	(*Robot At Home (Work Home or Intermediate Home)*)
	IF FB_In.Robot_Type=DX100
		THEN
		At_Home:= In_Cube64 OR In_Cube1 OR In_Cube2 OR In_Cube3 OR In_Cube4;
	ELSIF FB_In.Robot_Type=DX100_Dual
		THEN
		At_Home:= In_Cube64 OR In_Cube1 OR In_Cube2 OR In_Cube3 OR In_Cube4;
	ELSIF FB_In.Robot_Type=DX100_3_MIG
		THEN
		R1_At_Home:= R1_In_Cube64;
		R2_At_Home:= R2_In_Cube63;
		R3_At_Home:= R3_In_Cube62;
		At_Home:= R1_At_Home AND R2_At_Home AND R3_At_Home;
	ELSIF FB_In.Robot_Type=NX100
		THEN
		At_Home:= In_Cube32 OR In_Cube1 OR In_Cube2 OR In_Cube3 OR In_Cube4;
	ELSE
		At_Home:= In_Cube24 OR In_Cube1 OR In_Cube2 OR In_Cube3 OR In_Cube4;
	END_IF;
	(*At Equipment Interference Zones*)
	At_EquipInterf1:= NOT Clear_Of_EquipInterf1 AND Clear_Of_EquipInterf2 AND Clear_Of_EquipInterf3 AND Clear_Of_EquipInterf4
					AND Clear_Of_EquipInterf5 AND Clear_Of_EquipInterf6 AND Clear_Of_EquipInterf7 AND Clear_Of_EquipInterf8;
	At_EquipInterf2:= Clear_Of_EquipInterf1 AND NOT Clear_Of_EquipInterf2 AND Clear_Of_EquipInterf3 AND Clear_Of_EquipInterf4
					AND Clear_Of_EquipInterf5 AND Clear_Of_EquipInterf6 AND Clear_Of_EquipInterf7 AND Clear_Of_EquipInterf8;
	At_EquipInterf3:= Clear_Of_EquipInterf1 AND Clear_Of_EquipInterf2 AND NOT Clear_Of_EquipInterf3 AND Clear_Of_EquipInterf4
					AND Clear_Of_EquipInterf5 AND Clear_Of_EquipInterf6 AND Clear_Of_EquipInterf7 AND Clear_Of_EquipInterf8;
	At_EquipInterf4:= Clear_Of_EquipInterf1 AND Clear_Of_EquipInterf2 AND Clear_Of_EquipInterf3 AND NOT Clear_Of_EquipInterf4
					AND Clear_Of_EquipInterf5 AND Clear_Of_EquipInterf6 AND Clear_Of_EquipInterf7 AND Clear_Of_EquipInterf8;
	At_EquipInterf5:= Clear_Of_EquipInterf1 AND Clear_Of_EquipInterf2 AND Clear_Of_EquipInterf3 AND Clear_Of_EquipInterf4
					AND NOT Clear_Of_EquipInterf5 AND Clear_Of_EquipInterf6 AND Clear_Of_EquipInterf7 AND Clear_Of_EquipInterf8;
	At_EquipInterf6:= Clear_Of_EquipInterf1 AND Clear_Of_EquipInterf2 AND Clear_Of_EquipInterf3 AND Clear_Of_EquipInterf4
					AND Clear_Of_EquipInterf5 AND NOT Clear_Of_EquipInterf6 AND Clear_Of_EquipInterf7 AND Clear_Of_EquipInterf8;
	At_EquipInterf7:= Clear_Of_EquipInterf1 AND Clear_Of_EquipInterf2 AND Clear_Of_EquipInterf3 AND Clear_Of_EquipInterf4
					AND Clear_Of_EquipInterf5 AND Clear_Of_EquipInterf6 AND NOT Clear_Of_EquipInterf7 AND Clear_Of_EquipInterf8;
	At_EquipInterf8:= Clear_Of_EquipInterf1 AND Clear_Of_EquipInterf2 AND Clear_Of_EquipInterf3 AND Clear_Of_EquipInterf4
					AND Clear_Of_EquipInterf5 AND Clear_Of_EquipInterf6 AND Clear_Of_EquipInterf7 AND NOT Clear_Of_EquipInterf8;

	(*At Operator Interference Zones*)
	At_HumanInterf1:= NOT Clear_Of_HumanInterf1 AND Clear_Of_HumanInterf2 AND Clear_Of_HumanInterf3 AND Clear_Of_HumanInterf4
					AND Clear_Of_HumanInterf5 AND Clear_Of_HumanInterf6 AND Clear_Of_HumanInterf7 AND Clear_Of_HumanInterf8;
	At_HumanInterf2:= Clear_Of_HumanInterf1 AND NOT Clear_Of_HumanInterf2 AND Clear_Of_HumanInterf3 AND Clear_Of_HumanInterf4
					AND Clear_Of_HumanInterf5 AND Clear_Of_HumanInterf6 AND Clear_Of_HumanInterf7 AND Clear_Of_HumanInterf8;
	At_HumanInterf3:= Clear_Of_HumanInterf1 AND Clear_Of_HumanInterf2 AND NOT  Clear_Of_HumanInterf3 AND Clear_Of_HumanInterf4
					AND Clear_Of_HumanInterf5 AND Clear_Of_HumanInterf6 AND Clear_Of_HumanInterf7 AND Clear_Of_HumanInterf8;
	At_HumanInterf4:= Clear_Of_HumanInterf1 AND Clear_Of_HumanInterf2 AND Clear_Of_HumanInterf3 AND NOT Clear_Of_HumanInterf4
					AND Clear_Of_HumanInterf5 AND Clear_Of_HumanInterf6 AND Clear_Of_HumanInterf7 AND Clear_Of_HumanInterf8;
	At_HumanInterf5:= Clear_Of_HumanInterf1 AND Clear_Of_HumanInterf2 AND Clear_Of_HumanInterf3 AND Clear_Of_HumanInterf4
					AND NOT Clear_Of_HumanInterf5 AND Clear_Of_HumanInterf6 AND Clear_Of_HumanInterf7 AND Clear_Of_HumanInterf8;
	At_HumanInterf6:= Clear_Of_HumanInterf1 AND Clear_Of_HumanInterf2 AND Clear_Of_HumanInterf3 AND Clear_Of_HumanInterf4
					AND Clear_Of_HumanInterf5 AND NOT Clear_Of_HumanInterf6 AND Clear_Of_HumanInterf7 AND Clear_Of_HumanInterf8;
	At_HumanInterf7:= Clear_Of_HumanInterf1 AND Clear_Of_HumanInterf2 AND Clear_Of_HumanInterf3 AND Clear_Of_HumanInterf4
					AND Clear_Of_HumanInterf5 AND Clear_Of_HumanInterf6 AND NOT Clear_Of_HumanInterf7 AND Clear_Of_HumanInterf8;
	At_HumanInterf8:= Clear_Of_HumanInterf1 AND Clear_Of_HumanInterf2 AND Clear_Of_HumanInterf3 AND Clear_Of_HumanInterf4
					AND Clear_Of_HumanInterf5 AND Clear_Of_HumanInterf6 AND Clear_Of_HumanInterf7 AND NOT Clear_Of_HumanInterf8;

	(*Check Interference Zones*)
	OK_At_EquipInterf1:= FB_In.OK_ToEnter_EquipInterf1 OR Clear_Of_EquipInterf1;
	OK_At_EquipInterf2:= FB_In.OK_ToEnter_EquipInterf2 OR Clear_Of_EquipInterf2;
	OK_At_EquipInterf3:= FB_In.OK_ToEnter_EquipInterf3 OR Clear_Of_EquipInterf3;
	OK_At_EquipInterf4:= FB_In.OK_ToEnter_EquipInterf4 OR Clear_Of_EquipInterf4;
	OK_At_EquipInterf5:= FB_In.OK_ToEnter_EquipInterf5 OR Clear_Of_EquipInterf5;
	OK_At_EquipInterf6:= FB_In.OK_ToEnter_EquipInterf6 OR Clear_Of_EquipInterf6;
	OK_At_EquipInterf7:= FB_In.OK_ToEnter_EquipInterf7 OR Clear_Of_EquipInterf7;
	OK_At_EquipInterf8:= FB_In.OK_ToEnter_EquipInterf8 OR Clear_Of_EquipInterf8;
	OK_At_EquipInterfALL:= OK_At_EquipInterf1 AND OK_At_EquipInterf2 AND OK_At_EquipInterf3 AND OK_At_EquipInterf4
						 AND OK_At_EquipInterf5 AND OK_At_EquipInterf6 AND OK_At_EquipInterf7 AND OK_At_EquipInterf8;

	OK_At_HumanInterf1:= FB_In.OK_ToEnter_HumanInterf1 OR Clear_Of_HumanInterf1;
	OK_At_HumanInterf2:= FB_In.OK_ToEnter_HumanInterf2 OR Clear_Of_HumanInterf2;
	OK_At_HumanInterf3:= FB_In.OK_ToEnter_HumanInterf3 OR Clear_Of_HumanInterf3;
	OK_At_HumanInterf4:= FB_In.OK_ToEnter_HumanInterf4 OR Clear_Of_HumanInterf4;
	OK_At_HumanInterf5:= FB_In.OK_ToEnter_HumanInterf5 OR Clear_Of_HumanInterf5;
	OK_At_HumanInterf6:= FB_In.OK_ToEnter_HumanInterf6 OR Clear_Of_HumanInterf6;
	OK_At_HumanInterf7:= FB_In.OK_ToEnter_HumanInterf7 OR Clear_Of_HumanInterf7;
	OK_At_HumanInterf8:= FB_In.OK_ToEnter_HumanInterf8 OR Clear_Of_HumanInterf8;
	OK_At_HumanInterfALL:= OK_At_HumanInterf1 AND OK_At_HumanInterf2 AND OK_At_HumanInterf3 AND OK_At_HumanInterf4
							AND OK_At_HumanInterf5 AND OK_At_HumanInterf6 AND OK_At_HumanInterf7 AND OK_At_HumanInterf8;

	OK_At_RobotInterfs.0:= FB_In.OK_ToEnter_RobotInterfs.0 OR Clear_Of_RobotInterfs.0;
	OK_At_RobotInterfs.1:= FB_In.OK_ToEnter_RobotInterfs.1 OR Clear_Of_RobotInterfs.1;
	OK_At_RobotInterfs.2:= FB_In.OK_ToEnter_RobotInterfs.2 OR Clear_Of_RobotInterfs.2;
	OK_At_RobotInterfs.3:= FB_In.OK_ToEnter_RobotInterfs.3 OR Clear_Of_RobotInterfs.3;
	OK_At_RobotInterfs.4:= FB_In.OK_ToEnter_RobotInterfs.4 OR Clear_Of_RobotInterfs.4;
	OK_At_RobotInterfs.5:= FB_In.OK_ToEnter_RobotInterfs.5 OR Clear_Of_RobotInterfs.5;
	OK_At_RobotInterfs.6:= FB_In.OK_ToEnter_RobotInterfs.6 OR Clear_Of_RobotInterfs.6;
	OK_At_RobotInterfs.7:= FB_In.OK_ToEnter_RobotInterfs.7 OR Clear_Of_RobotInterfs.7;
	OK_At_RobotInterfsALL:= (Ok_At_RobotInterfs = 255);

	(*All Interference Zones OK*)
	All_Interfs_OK:= At_Home OR (OK_At_EquipInterfALL AND OK_At_HumanInterfALL AND OK_At_RobotInterfsAll);

	(*Robot Ready*)
	Ready:= Servos_Are_On AND In_Play AND In_Remote;

	(*Robot Acks Proper, FIX, EOAT, Model, and Task IDs *)
	Ack_ID_TMR.PT:=T#1.5S;
	Ack_ID_TMR();

	Fix_ID_Flt:= NOT At_Home AND Fix_ID_Ack<>FB_In.Fix_ID;
	EOAT_ID_Flt:= NOT At_Home AND EOAT_ID_Ack<>0; (*%%%%%% NEEDS FURTHER WORK for V2.1%%%%%%*)
	Model_ID_FLT:= NOT At_Home AND Model_ID_Ack<> FB_In.Model_ID;
	Task_ID_Flt:= NOT At_Home AND Task_ID_Ack<250 AND (Task_ID_Ack<>FB_In.Task_ID OR Task_ID_Ack=0);

	(*If Fault Timer hasn't been triggered, ID Acks Are OK*)
	Ack_ID_TMR.IN:= Fix_ID_FLT OR EOAT_ID_FLT OR Model_ID_FLT OR Task_ID_FLT ;
	ID_Acks_OK:= NOT Ack_ID_TMR.Q;


	(*Turn On Servo Motors*)
	Servos_Req_Delay.PT:=T#1.25s;
	Servos_Req_Delay();
	Servos_Req_Delay.IN:= Estop_Relays_On AND SafetyGate_Relays_On AND In_Remote AND In_Play AND NOT Faulted AND NOT Servos_Are_On;
	Servos_Req:= Servos_Req_Delay.Q;

	(*Turn Servo Motors Off*)
	IF NOT ID_Acks_OK AND NOT In_Teach AND NOT At_Home
		THEN Servos_Off_Req:= TRUE;
	ELSE Servos_Off_Req:= FALSE;
	END_IF;
	IF NOT Estop_Relays_On OR NOT FB_In.Teach_Interlock
		THEN Servos_Off_Req:= TRUE;
	ELSE Servos_Off_Req:= FALSE;
	END_IF;

	(*Start Robot Scan*)
	(*%%%%%%%%%% WOULD LIKE TO CLEAN UP A LITTLE %%%%%%%%%%%*)
	IF (FB_In.Start_Scan OR Robot_Is_AutoRestart) AND NOT FB_In.Stop_Scan2 AND Ready AND Estop_Relays_On AND SafetyGate_Relays_On AND All_Interfs_OK
		THEN
		IF At_Home OR ID_Acks_OK
			THEN
				Start_Robot_Scan:=FB_In.Start_Scan;
		END_IF;
	ELSE
		Start_Robot_Scan:=FALSE;
	END_IF;

	(*Hold Robot*)
	(*%%%%%%%%%% WOULD LIKE TO CLEAN UP A LITTLE %%%%%%%%%%%*)
	IF Estop_Relays_On AND FB_IN.Enable_Motion AND NOT FB_In.Stop_Scan AND NOT FB_In.Stop_Scan2
		THEN
		IF In_Teach
			THEN
				Hold_Robot:= FALSE;
		ELSIF (At_Home OR
				(Task_ID_Ack<>0 AND (Fix_ID_Ack<>0 OR Task_ID_Ack>250) AND ID_Acks_OK AND All_Interfs_OK))
				AND SafetyGate_Relays_On  AND Collision_Detect_Valid AND NOT FB_In.Major_Faults
			THEN
				Hold_Robot:=FALSE;
		ELSE
				Hold_Robot:= TRUE;
		END_IF;
	ELSE
		Hold_Robot:= TRUE;
	END_IF;

(*Troubleshooting Code*)
IF NOT Estop_Relays_On
	THEN Temp1:= TRUE;
END_IF;
IF NOT FB_In.Enable_Motion
	THEN Temp2:= TRUE;
END_IF;
IF FB_In.Stop_Scan
	THEN Temp3:= TRUE;
END_IF;
IF NOT At_Home
	THEN Temp4:= TRUE;
END_IF;
IF NOT ID_Acks_OK
	THEN Temp5:= TRUE;
END_IF;
IF NOT All_Interfs_OK
	THEN Temp6:= TRUE;
END_IF;
IF NOT SafetyGate_Relays_On
	THEN Temp7:= TRUE;
END_IF;
IF NOT Collision_Detect_Valid
	THEN Temp8:= TRUE;
END_IF;
IF FB_In.Safety_RST
	THEN
		Temp1:= FALSE;
		Temp2:= FALSE;
		Temp3:= FALSE;
		Temp4:= FALSE;
		Temp5:= FALSE;
		Temp6:= FALSE;
		Temp7:= FALSE;
		Temp8:= FALSE;
END_IF;

(*$$$$$$$$$$$$$$$$$$$$$$$$$$$$$$$$$$$$$$$$$$$$$ Status Banner $$$$$$$$$$$$$$$$$$$$$$$$$$$$$$$$$$$$$$$$$$$$$$$$$$$$$$$$$$*)
	(*Mesages 1 through 9 are reserved for legacy code*)
	(*Spare*)
	IF FALSE
		THEN Status:= 1;
	(*Spare*)
	ELSIF FALSE
		THEN Status:= 2;
	(*Spare*)
	ELSIF FALSE
		THEN Status:= 3;
	(*Spare*)
	ELSIF FALSE
		THEN Status:= 4;
	(*Robot Home and Ready*)
	ELSIF At_Home AND Operating AND NOT Faulted AND NOT Ack_ID_Flt AND Task_ID_Ack=0
		THEN Status:= 10;
	(*Robot Waiting For Start*)
	ELSIF  Ready AND NOT Operating AND NOT Faulted AND ID_Acks_OK
		THEN Status:= 11;
	(*Robot Servos Not On*)
	ELSIF NOT Ready AND NOT Servos_Are_On AND In_Remote AND In_Play AND NOT In_Teach AND NOT Faulted AND ID_Acks_OK
		THEN Status:= 14;
	(*Robot Not In Play*)
	ELSIF NOT Ready AND In_Remote AND NOT In_Play AND NOT In_Teach AND NOT Faulted AND ID_Acks_OK
		THEN Status:= 15;
	(*Robot Not In Remote*)
	ELSIF NOT Ready AND NOT In_Remote AND In_Play AND NOT In_Teach AND NOT Faulted AND ID_Acks_OK
		THEN Status:= 16;
	(*Robot In Teach*)
	ELSIF  NOT Ready AND (NOT In_Remote OR FB_In.Robot_Type=XRC) AND NOT In_Play AND In_Teach AND NOT Faulted AND ID_Acks_OK
		THEN Status:= 17;
	(*Robot Held by Teach Interlock*)
	ELSIF NOT FB_In.Teach_Interlock
		THEN Status:= 30;
	(*Robot Faulted*)
	ELSIF Faulted
		THEN Status:= 31;
	(*Robot Fix Id Ack Fault*)
	ELSIF NOT ID_Acks_OK AND Fix_ID_Flt
		THEN Status:= 32;
	(*Robot EOAT Id Ack Fault*)
	ELSIF NOT ID_Acks_OK AND EOAT_ID_Flt
		THEN Status:= 33;
	(*Robot Task Id Ack Fault*)
	ELSIF NOT ID_Acks_OK AND Task_ID_Flt
		THEN Status:= 34;
	(*Robot Custom Messages (See Global Variables, Task ID Record) *)
	ELSIF (NOT At_Home OR Task_ID_Ack=255) AND Task_Id_Ack<>0 AND Ready AND Operating AND NOT Faulted AND ID_Acks_OK
		THEN Status:= Task_ID_Ack+100;
	(*Produce "Invalid Data" If None of The Above Hold True To Blank Status Banner, but only if not at Home*)
	ELSE
		IF NOT At_Home
		 THEN
			Status:=0;
		END_IF;
	END_IF;
(*$$$$$$$$$$$$$$$$$$$$$$$$$$$$$$$$$$$$$$$$$$$$$$$$$$$ Faults $$$$$$$$$$$$$$$$$$$$$$$$$$$$$$$$$$$$$$$$$$$$$$$$$$$$$$$*)

(*$$$$$$$$$$$$$$$$$$$$$$$$$$$$$$$$$$$$$$$$$$$$$$ Transfer Standard Outputs $$$$$$$$$$$$$$$$$$$$$$$$$$$$$$$$$$$$$$$$$$$*)
	(*Transfer I/O Images for Display On HMI*)
	Input_Image:=In_From_HW;
	Output_Image:=Out_To_HW;

	Discrete_Image.T01:=T01;
	Discrete_Image.T02_STAT:=T02_STAT;
	Discrete_Image.T03:=T03;
	Discrete_Image.T04:=T04;
	Discrete_Image.T05:=T05;
	Discrete_Image.T06:=T06;
	Discrete_Image.T07:=T07;
	Discrete_Image.T08:=T08;
	Discrete_Image.T09:=T09;
	Discrete_Image.T10:=T10;


	(*Transfer Commands to ECAT Outputs*)
	Out_To_ECAT.SYS.0:= Start_Robot_Scan;			(*Start Robot Scan*)
	Out_To_ECAT.SYS.1:= Servos_Req;				(*Turn on Servos*)
	Out_To_ECAT.SYS.2:= FALSE;					(*Master Job Call*)
	Out_To_ECAT.SYS.3:= FB_In.Alarm_RST;			(*Alarm Reset*)
	IF FB_In.Robot_Type=NX100 OR FB_In.Robot_Type=DX100 OR FB_In.Robot_Type=DX100_Dual
		THEN
			Out_To_ECAT.SYS.4:= FALSE;					(*Undefined*)
				Play_Delay.PT:=T#0.5S;
				Play_Delay.IN:= In_Remote;
			Out_To_ECAT.SYS.5:= Play_Delay.Q;				(*Play Mode Select*)
			IF FB_In.Robot_Type=DX100 OR FB_In.Robot_Type=DX100_Dual
				THEN
					Out_To_ECAT.SYS.6:= FB_In.Select_Teach;					(*Select Teach Mode*)
			ELSIF FB_In.Robot_Type=NX100
				THEN
				Out_To_ECAT.SYS.6:= Servos_Off_Req;					(*Select Teach Mode*)
			END_IF;
	ELSE
			Out_To_ECAT.SYS.4:= FB_In.Select_Remote;		(*Select Remote Mode*)
			Out_To_ECAT.SYS.5:= FB_In.Select_Play;			(*Select Play Mode*)
			Out_To_ECAT.SYS.6:= FB_In.Select_Teach;		(*Select Teach Mode*)
	END_IF;

	Out_To_ECAT.SYS.7:= Hold_Robot;						(*Hold Robot, (N.O. IE; High to Hold)*)


	Out_To_ECAT.SYS.8:= FALSE;							(*Cube 1 Entrance Prohibit*)
	Out_To_ECAT.SYS.9:= FALSE;							(*Cube 2 Entrance Prohibit*)
	Out_To_ECAT.SYS.10:= FB_In.Weld_Inhibit;				(*Weld Inhibit (Current Only)*)
	Out_To_ECAT.SYS.11:= FALSE;							(*Weld Stop (Gun and Current)*)
	Out_To_ECAT.SYS.12:= FALSE;							(*Cube 3 Entrance Prohibit*)

	IF FB_In.Robot_Type=DX100_3_MIG
		THEN Out_To_ECAT.SYS.13:= FB_In.Low_Speed;		(*Low Speed Mode DX100_3_MIG*)
	ELSE
			Out_To_ECAT.SYS.13:= FALSE;					(*Cube 4 Entrance Prohibit*)
	END_IF;

	IF NOT (FB_In.Robot_Type=DX100_3_MIG)
		THEN Out_To_ECAT.SYS.14:= FB_In.Low_Speed;		(*Safety Speed Select*)
	ELSE
			Out_To_ECAT.SYS.14:= FALSE;
	END_IF;

	IF FB_In.Robot_Type=XRC
		THEN
			Out_To_ECAT.SYS.15:= Servos_Off_Req;			(*Turns Off Servo Motors*)
	ELSE
			Out_To_ECAT.SYS.15:= FALSE;					(*Undefined*)
	END_IF;


	(*IG#4*)
	Out_To_ECAT.IG4.0:= TRUE;								(*True = turntable and robots enabled, False= turntable only*)
	Out_To_ECAT.IG4.1:= FALSE;								(*Robot Sweep Cycle Start*)
	Out_To_ECAT.IG4.2:= T05.I.2 AND T04.I.0 AND T04.I.1;			(*Light curtain Clear (Substituted with External Axis Enabled)*)
	Out_To_ECAT.IG4.3:= Table_SideA_At_Robots;				(*Turntable (Ext Axis S1), Side A at Robots*)
	Out_To_ECAT.IG4.4:= Table_SideB_At_Robots;				(*Turntable (Ext Axis S1), Side B at Robots*)
	Out_To_ECAT.IG4.5:= FALSE;								(*Spare*)
	Out_To_ECAT.IG4.6:= FALSE; 		 						(*Spare*)
	Out_To_ECAT.IG4.7:= FALSE;  								(*Spare*)

	(*IG#5*)
	Out_To_ECAT.IG5.0:= FALSE;								(*Spare*)
	Out_To_ECAT.IG5.1:= FALSE;								(*Spare*)
	Out_To_ECAT.IG5.2:= FALSE;								(*Spare*)
	Out_To_ECAT.IG5.3:= FALSE;								(*Spare*)
	Out_To_ECAT.IG5.4:= FALSE;								(*Spare*)
	Out_To_ECAT.IG5.5:= FALSE;								(*Spare*)
	Out_To_ECAT.IG5.6:= FALSE; 		 						(*Spare*)
	Out_To_ECAT.IG5.7:= FALSE;  								(*Spare*)
	(*IG#6*)
	Out_To_ECAT.IG6.0:= FB_In.OK_ToEnter_EquipInterf1;			(*OK to Enter Equip Interf Zone#1*)
	Out_To_ECAT.IG6.1:= FB_In.OK_ToEnter_EquipInterf2;			(*OK to Enter Equip Interf Zone#2*)
	Out_To_ECAT.IG6.2:= FB_In.OK_ToEnter_EquipInterf3;			(*OK to Enter Equip Interf Zone#3*)
	Out_To_ECAT.IG6.3:= FB_In.OK_ToEnter_EquipInterf4;			(*OK to Enter Equip Interf Zone#4*)
	Out_To_ECAT.IG6.4:= FB_In.OK_ToEnter_EquipInterf5;			(*OK to Enter Equip Interf Zone#1*)
	Out_To_ECAT.IG6.5:= FB_In.OK_ToEnter_EquipInterf6;			(*OK to Enter Equip Interf Zone#2*)
	Out_To_ECAT.IG6.6:= FB_In.OK_ToEnter_EquipInterf7;			(*OK to Enter Equip Interf Zone#3*)
	Out_To_ECAT.IG6.7:= FB_In.OK_ToEnter_EquipInterf8;			(*OK to Enter Equip Interf Zone#4*)
	(*IG#7*)
	Out_To_ECAT.IG7.0:= FB_In.OK_ToEnter_HumanInterf1;			(*OK to Enter Human Interf Zone#1*)
	Out_To_ECAT.IG7.1:= FB_In.OK_ToEnter_HumanInterf2;			(*OK to Enter Human Interf Zone#2*)
	Out_To_ECAT.IG7.2:= FB_In.OK_ToEnter_HumanInterf3;			(*OK to Enter Human Interf Zone#3*)
	Out_To_ECAT.IG7.3:= FB_In.OK_ToEnter_HumanInterf4;			(*OK to Enter Human Interf Zone#4*)
	Out_To_ECAT.IG7.4:= FB_In.OK_ToEnter_HumanInterf5;			(*OK to Enter Human Interf Zone#5*)
	Out_To_ECAT.IG7.5:= FB_In.OK_ToEnter_HumanInterf6;			(*OK to Enter Human Interf Zone#6*)
	Out_To_ECAT.IG7.6:= FB_In.OK_ToEnter_HumanInterf7;			(*OK to Enter Human Interf Zone#7*)
	Out_To_ECAT.IG7.7:= FB_In.OK_ToEnter_HumanInterf8;			(*OK to Enter Human Interf Zone#8*)
	(*IG#8*)
	Out_To_ECAT.IG8:= UDINT_TO_BYTE(FB_In.EOAT_ID);									(*EOAT_ID*)
	(*IG#9*)
	IF Task_ID_Ack<>0 AND Task_ID_Ack=FB_In.Task_ID
		THEN
			Out_To_ECAT.IG9:= UINT_TO_BYTE(FB_In.Fix_ID);								(*Fix_ID*)
	ELSE
			Out_To_ECAT.IG9:=0;
	END_IF;
	(*IG#10*)
	Out_To_ECAT.IG10:= UINT_TO_BYTE(FB_In.Model_ID);									(*Model_ID*)
	(*IG#11*)
	Out_To_ECAT.IG11:= UINT_TO_BYTE(FB_In.Task_ID);										(*Task_ID*)
	(*IG#12*)
	Out_To_ECAT.IG12.0:= Peripheral_Req.0 AND FB_In.PeripheralReq_Ack.0;						(*Peripheral Equipment Request 1 (Reposition request etc.)*)
	Out_To_ECAT.IG12.1:= Peripheral_Req.1 AND FB_In.PeripheralReq_Ack.1;						(*Peripheral Equipment Request 2 (Reposition request etc.)*)
	Out_To_ECAT.IG12.2:= Peripheral_Req.2 AND FB_In.PeripheralReq_Ack.2;						(*Peripheral Equipment Request 4 (Reposition request etc.)*)
	Out_To_ECAT.IG12.3:= Peripheral_Req.3 AND FB_In.PeripheralReq_Ack.3;						(*Peripheral Equipment Request 8 (Reposition request etc.)*)
	Out_To_ECAT.IG12.4:= Peripheral_Req.4 AND FB_In.PeripheralReq_Ack.4;						(*Peripheral Equipment Request 16 (Reposition request etc.)*)
	Out_To_ECAT.IG12.5:= Peripheral_Req.5 AND FB_In.PeripheralReq_Ack.5;						(*Peripheral Equipment Request 32 (Reposition request etc.)*)
	Out_To_ECAT.IG12.6:= Peripheral_Req.6 AND FB_In.PeripheralReq_Ack.6;						(*Peripheral Equipment Request 64 (Reposition request etc.)*)
	Out_To_ECAT.IG12.7:= Peripheral_Req.7 AND FB_In.PeripheralReq_Ack.7;						(*Peripheral Equipment Request 128 (Reposition request etc.)*)
	(*IG#13*)
	IF At_Pounce AND Task_ID_Ack<>0 AND Task_ID_Ack=FB_In.Task_ID AND Fix_Id_Ack<>0 AND Fix_ID_Ack=FB_In.Fix_ID
		THEN
			Out_To_ECAT.IG13.0:= FB_In.Proceed_From_Pounce;		(*Proceed >From Pounce*)
	ELSE
			Out_To_ECAT.IG13.0:= FALSE;						(*Proceed From Pounce*)
	END_IF;
	Out_To_ECAT.IG13.3:= FALSE;										(*Spare*)
	Out_To_ECAT.IG13.3:= Clear_To_Unclamp;							(*Robot is Clear for Tool to Unclamp Early Ack*)
	Out_To_ECAT.IG13.7:= Task_Completed AND FB_In.Complete_Ack;					(*Task Completed Ack*)

	(*IG#14*)
	Out_To_ECAT.IG14.0:= Fb_In.OK_ToEnter_RobotInterfs.0;
	Out_To_ECAT.IG14.1:= Fb_In.OK_ToEnter_RobotInterfs.1;
	Out_To_ECAT.IG14.2:= Fb_In.OK_ToEnter_RobotInterfs.2;
	Out_To_ECAT.IG14.3:= Fb_In.OK_ToEnter_RobotInterfs.3;
	Out_To_ECAT.IG14.4:= Fb_In.OK_ToEnter_RobotInterfs.4;
	Out_To_ECAT.IG14.5:= Fb_In.OK_ToEnter_RobotInterfs.5;
	Out_To_ECAT.IG14.6:= Fb_In.OK_ToEnter_RobotInterfs.6;
	Out_To_ECAT.IG14.7:= Fb_In.OK_ToEnter_RobotInterfs.7;

	(*IG#17*)
	Out_To_ECAT.IG17.0:= EOAT_Req.0 AND FB_In.EOATReq_Ack.0;						(*EOAT Request 1 (Reposition request etc.)*)
	Out_To_ECAT.IG17.1:= EOAT_Req.1 AND FB_In.EOATReq_Ack.1;						(*EOAT Request 2 (Reposition request etc.)*)
	Out_To_ECAT.IG17.2:= EOAT_Req.2 AND FB_In.EOATReq_Ack.2;						(*EOAT Request 4 (Reposition request etc.)*)
	Out_To_ECAT.IG17.3:= EOAT_Req.3 AND FB_In.EOATReq_Ack.3;						(*EOAT Request 8 (Reposition request etc.)*)
	Out_To_ECAT.IG17.4:= EOAT_Req.4 AND FB_In.EOATReq_Ack.4;						(*EOAT Request 16 (Reposition request etc.)*)
	Out_To_ECAT.IG17.5:= EOAT_Req.5 AND FB_In.EOATReq_Ack.5;						(*EOAT Request 32 (Reposition request etc.)*)
	Out_To_ECAT.IG17.6:= EOAT_Req.6 AND FB_In.EOATReq_Ack.6;						(*EOAT Request 64 (Reposition request etc.)*)
	Out_To_ECAT.IG17.7:= EOAT_Req.7 AND FB_In.EOATReq_Ack.7;						(*EOAT Request 128 (Reposition request etc.)*)

(*----------------- Gather KUKA Type Data and convert to Generic Robot Type for Transfer to Output Image*)

Out_To_HW:= FUN_GTAC_MOTOMAN32_TO_GenericRobotOutputImage(Out_To_ECAT);

(*$$$$$$$$$$$$$$$$$$$$$$$$$$$$$$$$$$$$$$$$$$$$$$$ Transfer Safety Outputs $$$$$$$$$$$$$$$$$$$$$$$$$$$$$$$$$$$$$$$$$$$$$$$*)
	(*Set All Safety Groups to Run*)
		T02_CMD.SGs_RUNSTOP:= TRUE;
	(*Reset Of Safety Group Errors*)
		T02_CMD.SGs_ERRAck:= FB_In.Safety_RST;
	(*Reset Only Used FBs With In Safety Group*)
		(*Reset of Estop, Safety Gate and Misc FBs*)
		T02_CMD.FBs_ControlPowerPB:= FB_In.Safety_RST;

END_FUNCTION_BLOCK

// ---- POUs/FUNs/FUN_GTAC_GenericRobotInputImage_TO_MOTOMAN32.TcPOU
(*Function used to map HW Byte Array Typed Generic Input Image (from Robot Outputs) to Motoman 32 Byte Profibus Interface Type
to more closly ressemble Robot Output structure in teach pendant
	author: Brent Lekx-Toniolo of Sodecia GTAC
	date: November 2012
------------------------------------------------------------------------------------------
REVISION NOTES:
	version 1.0
		- initial concept

	- 20151105
		- Changed type for conversion of Motoman to Ethercat, b.lekx-toniolo

------------------------------------------------------------------------------------------
*)

FUNCTION FUN_GTAC_GenericRobotInputImage_TO_MOTOMAN32 : udt_EtherCAT_Motoman_Input_20151105
VAR_INPUT
	ByteBased_Array: udt_GenericRobot_AnyFieldbus_InputBytes_20220421;
END_VAR
VAR
END_VAR

(*Gathering of Generic Byte Typed Array to map to Robot Specific Data Type Points*)
			(*Map System Section*)
			FUN_GTAC_GenericRobotInputImage_TO_MOTOMAN32.SYS.0:= ByteBased_Array.Byte_[1].0;
			FUN_GTAC_GenericRobotInputImage_TO_MOTOMAN32.SYS.1:= ByteBased_Array.Byte_[1].1;
			FUN_GTAC_GenericRobotInputImage_TO_MOTOMAN32.SYS.2:= ByteBased_Array.Byte_[1].2;
			FUN_GTAC_GenericRobotInputImage_TO_MOTOMAN32.SYS.3:= ByteBased_Array.Byte_[1].3;
			FUN_GTAC_GenericRobotInputImage_TO_MOTOMAN32.SYS.4:= ByteBased_Array.Byte_[1].4;
			FUN_GTAC_GenericRobotInputImage_TO_MOTOMAN32.SYS.5:= ByteBased_Array.Byte_[1].5;
			FUN_GTAC_GenericRobotInputImage_TO_MOTOMAN32.SYS.6:= ByteBased_Array.Byte_[1].6;
			FUN_GTAC_GenericRobotInputImage_TO_MOTOMAN32.SYS.7:= ByteBased_Array.Byte_[1].7;

			FUN_GTAC_GenericRobotInputImage_TO_MOTOMAN32.SYS.8:= ByteBased_Array.Byte_[2].0;
			FUN_GTAC_GenericRobotInputImage_TO_MOTOMAN32.SYS.9:= ByteBased_Array.Byte_[2].1;
			FUN_GTAC_GenericRobotInputImage_TO_MOTOMAN32.SYS.10:= ByteBased_Array.Byte_[2].2;
			FUN_GTAC_GenericRobotInputImage_TO_MOTOMAN32.SYS.11:= ByteBased_Array.Byte_[2].3;
			FUN_GTAC_GenericRobotInputImage_TO_MOTOMAN32.SYS.12:= ByteBased_Array.Byte_[2].4;
			FUN_GTAC_GenericRobotInputImage_TO_MOTOMAN32.SYS.13:= ByteBased_Array.Byte_[2].5;
			FUN_GTAC_GenericRobotInputImage_TO_MOTOMAN32.SYS.14:= ByteBased_Array.Byte_[2].6;
			FUN_GTAC_GenericRobotInputImage_TO_MOTOMAN32.SYS.15:= ByteBased_Array.Byte_[2].7;

			(*Map Standard Section*)
			FUN_GTAC_GenericRobotInputImage_TO_MOTOMAN32.OG4:= ByteBased_Array.Byte_[3];
			FUN_GTAC_GenericRobotInputImage_TO_MOTOMAN32.OG5:= ByteBased_Array.Byte_[4];
			FUN_GTAC_GenericRobotInputImage_TO_MOTOMAN32.OG6:= ByteBased_Array.Byte_[5];
			FUN_GTAC_GenericRobotInputImage_TO_MOTOMAN32.OG7:= ByteBased_Array.Byte_[6];
			FUN_GTAC_GenericRobotInputImage_TO_MOTOMAN32.OG8:= ByteBased_Array.Byte_[7];
			FUN_GTAC_GenericRobotInputImage_TO_MOTOMAN32.OG9:= ByteBased_Array.Byte_[8];
			FUN_GTAC_GenericRobotInputImage_TO_MOTOMAN32.OG10:= ByteBased_Array.Byte_[9];
			FUN_GTAC_GenericRobotInputImage_TO_MOTOMAN32.OG11:= ByteBased_Array.Byte_[10];
			FUN_GTAC_GenericRobotInputImage_TO_MOTOMAN32.OG12:= ByteBased_Array.Byte_[11];
			FUN_GTAC_GenericRobotInputImage_TO_MOTOMAN32.OG13:= ByteBased_Array.Byte_[12];
			FUN_GTAC_GenericRobotInputImage_TO_MOTOMAN32.OG14:= ByteBased_Array.Byte_[13];
			FUN_GTAC_GenericRobotInputImage_TO_MOTOMAN32.OG15:= ByteBased_Array.Byte_[14];
			FUN_GTAC_GenericRobotInputImage_TO_MOTOMAN32.OG16:= ByteBased_Array.Byte_[15];
			FUN_GTAC_GenericRobotInputImage_TO_MOTOMAN32.OG17:= ByteBased_Array.Byte_[16];
			FUN_GTAC_GenericRobotInputImage_TO_MOTOMAN32.OG18:= ByteBased_Array.Byte_[17];
			FUN_GTAC_GenericRobotInputImage_TO_MOTOMAN32.OG19:= ByteBased_Array.Byte_[18];
			FUN_GTAC_GenericRobotInputImage_TO_MOTOMAN32.OG20:= ByteBased_Array.Byte_[19];
			FUN_GTAC_GenericRobotInputImage_TO_MOTOMAN32.OG21:= ByteBased_Array.Byte_[20];
			FUN_GTAC_GenericRobotInputImage_TO_MOTOMAN32.OG22:= ByteBased_Array.Byte_[21];
			FUN_GTAC_GenericRobotInputImage_TO_MOTOMAN32.OG23:= ByteBased_Array.Byte_[22];
			FUN_GTAC_GenericRobotInputImage_TO_MOTOMAN32.OG24:= ByteBased_Array.Byte_[23];
			FUN_GTAC_GenericRobotInputImage_TO_MOTOMAN32.OG25:= ByteBased_Array.Byte_[24];
			FUN_GTAC_GenericRobotInputImage_TO_MOTOMAN32.OG26:= ByteBased_Array.Byte_[25];
			FUN_GTAC_GenericRobotInputImage_TO_MOTOMAN32.OG27:= ByteBased_Array.Byte_[26];
			FUN_GTAC_GenericRobotInputImage_TO_MOTOMAN32.OG28:= ByteBased_Array.Byte_[27];
			FUN_GTAC_GenericRobotInputImage_TO_MOTOMAN32.OG29:= ByteBased_Array.Byte_[28];
			FUN_GTAC_GenericRobotInputImage_TO_MOTOMAN32.OG30:= ByteBased_Array.Byte_[29];
			FUN_GTAC_GenericRobotInputImage_TO_MOTOMAN32.OG31:= ByteBased_Array.Byte_[30];
			FUN_GTAC_GenericRobotInputImage_TO_MOTOMAN32.OG32:= ByteBased_Array.Byte_[31];
			FUN_GTAC_GenericRobotInputImage_TO_MOTOMAN32.OG33:= ByteBased_Array.Byte_[32];

END_FUNCTION

// ---- POUs/FUNs/FUN_GTAC_MOTOMAN32_TO_GenericRobotOutputImage.TcPOU
(*Function used to map Motoman 32 Byte Profibus Interface Type to HW Byte Array Typed Generic Output Image (to Robot Inputs)
to more closly ressemble Robot Input structure in teach pendant
	author: Brent Lekx-Toniolo of Sodecia GTAC
	date: November 2012
------------------------------------------------------------------------------------------
REVISION NOTES:

	version 1
		- initial concept
	- 20151105
		- Changed type for conversion of Motoman to Ethercat, b.lekx-toniolo

-------------------------------------------------------------------------------------------
*)

FUNCTION FUN_GTAC_MOTOMAN32_TO_GenericRobotOutputImage : udt_GenericRobot_AnyFieldbus_OutputBytes_20220421
VAR_INPUT
	Motoman32_Typed_Data: udt_EtherCAT_Motoman_Output_20151105;
END_VAR
VAR
END_VAR

(*Gathering of Robot Specific Data Type Points to Map to Generic Byte Typed Array*)
			(*Map System Section*)
			FUN_GTAC_MOTOMAN32_TO_GenericRobotOutputImage.Byte_[1].0:= Motoman32_Typed_Data.SYS.0;
			FUN_GTAC_MOTOMAN32_TO_GenericRobotOutputImage.Byte_[1].1:= Motoman32_Typed_Data.SYS.1;
			FUN_GTAC_MOTOMAN32_TO_GenericRobotOutputImage.Byte_[1].2:= Motoman32_Typed_Data.SYS.2;
			FUN_GTAC_MOTOMAN32_TO_GenericRobotOutputImage.Byte_[1].3:= Motoman32_Typed_Data.SYS.3;
			FUN_GTAC_MOTOMAN32_TO_GenericRobotOutputImage.Byte_[1].4:= Motoman32_Typed_Data.SYS.4;
			FUN_GTAC_MOTOMAN32_TO_GenericRobotOutputImage.Byte_[1].5:= Motoman32_Typed_Data.SYS.5;
			FUN_GTAC_MOTOMAN32_TO_GenericRobotOutputImage.Byte_[1].6:= Motoman32_Typed_Data.SYS.6;
			FUN_GTAC_MOTOMAN32_TO_GenericRobotOutputImage.Byte_[1].7:= Motoman32_Typed_Data.SYS.7;

			FUN_GTAC_MOTOMAN32_TO_GenericRobotOutputImage.Byte_[2].0:= Motoman32_Typed_Data.SYS.8;
			FUN_GTAC_MOTOMAN32_TO_GenericRobotOutputImage.Byte_[2].1:= Motoman32_Typed_Data.SYS.9;
			FUN_GTAC_MOTOMAN32_TO_GenericRobotOutputImage.Byte_[2].2:= Motoman32_Typed_Data.SYS.10;
			FUN_GTAC_MOTOMAN32_TO_GenericRobotOutputImage.Byte_[2].3:= Motoman32_Typed_Data.SYS.11;
			FUN_GTAC_MOTOMAN32_TO_GenericRobotOutputImage.Byte_[2].4:= Motoman32_Typed_Data.SYS.12;
			FUN_GTAC_MOTOMAN32_TO_GenericRobotOutputImage.Byte_[2].5:= Motoman32_Typed_Data.SYS.13;
			FUN_GTAC_MOTOMAN32_TO_GenericRobotOutputImage.Byte_[2].6:= Motoman32_Typed_Data.SYS.14;
			FUN_GTAC_MOTOMAN32_TO_GenericRobotOutputImage.Byte_[2].7:= Motoman32_Typed_Data.SYS.15;

			(*Map Standard Section*)
			FUN_GTAC_MOTOMAN32_TO_GenericRobotOutputImage.Byte_[3]:= Motoman32_Typed_Data.IG4;
			FUN_GTAC_MOTOMAN32_TO_GenericRobotOutputImage.Byte_[4]:= Motoman32_Typed_Data.IG5;
			FUN_GTAC_MOTOMAN32_TO_GenericRobotOutputImage.Byte_[5]:= Motoman32_Typed_Data.IG6;
			FUN_GTAC_MOTOMAN32_TO_GenericRobotOutputImage.Byte_[6]:= Motoman32_Typed_Data.IG7;
			FUN_GTAC_MOTOMAN32_TO_GenericRobotOutputImage.Byte_[7]:= Motoman32_Typed_Data.IG8;
			FUN_GTAC_MOTOMAN32_TO_GenericRobotOutputImage.Byte_[8]:= Motoman32_Typed_Data.IG9;
			FUN_GTAC_MOTOMAN32_TO_GenericRobotOutputImage.Byte_[9]:= Motoman32_Typed_Data.IG10;
			FUN_GTAC_MOTOMAN32_TO_GenericRobotOutputImage.Byte_[10]:= Motoman32_Typed_Data.IG11;
			FUN_GTAC_MOTOMAN32_TO_GenericRobotOutputImage.Byte_[11]:= Motoman32_Typed_Data.IG12;
			FUN_GTAC_MOTOMAN32_TO_GenericRobotOutputImage.Byte_[12]:= Motoman32_Typed_Data.IG13;
			FUN_GTAC_MOTOMAN32_TO_GenericRobotOutputImage.Byte_[13]:= Motoman32_Typed_Data.IG14;
			FUN_GTAC_MOTOMAN32_TO_GenericRobotOutputImage.Byte_[14]:= Motoman32_Typed_Data.IG15;
			FUN_GTAC_MOTOMAN32_TO_GenericRobotOutputImage.Byte_[15]:= Motoman32_Typed_Data.IG16;
			FUN_GTAC_MOTOMAN32_TO_GenericRobotOutputImage.Byte_[16]:= Motoman32_Typed_Data.IG17;
			FUN_GTAC_MOTOMAN32_TO_GenericRobotOutputImage.Byte_[17]:= Motoman32_Typed_Data.IG18;
			FUN_GTAC_MOTOMAN32_TO_GenericRobotOutputImage.Byte_[18]:= Motoman32_Typed_Data.IG19;
			FUN_GTAC_MOTOMAN32_TO_GenericRobotOutputImage.Byte_[19]:= Motoman32_Typed_Data.IG20;
			FUN_GTAC_MOTOMAN32_TO_GenericRobotOutputImage.Byte_[20]:= Motoman32_Typed_Data.IG21;
			FUN_GTAC_MOTOMAN32_TO_GenericRobotOutputImage.Byte_[21]:= Motoman32_Typed_Data.IG22;
			FUN_GTAC_MOTOMAN32_TO_GenericRobotOutputImage.Byte_[22]:= Motoman32_Typed_Data.IG23;
			FUN_GTAC_MOTOMAN32_TO_GenericRobotOutputImage.Byte_[23]:= Motoman32_Typed_Data.IG24;
			FUN_GTAC_MOTOMAN32_TO_GenericRobotOutputImage.Byte_[24]:= Motoman32_Typed_Data.IG25;
			FUN_GTAC_MOTOMAN32_TO_GenericRobotOutputImage.Byte_[25]:= Motoman32_Typed_Data.IG26;
			FUN_GTAC_MOTOMAN32_TO_GenericRobotOutputImage.Byte_[26]:= Motoman32_Typed_Data.IG27;
			FUN_GTAC_MOTOMAN32_TO_GenericRobotOutputImage.Byte_[27]:= Motoman32_Typed_Data.IG28;
			FUN_GTAC_MOTOMAN32_TO_GenericRobotOutputImage.Byte_[28]:= Motoman32_Typed_Data.IG29;
			FUN_GTAC_MOTOMAN32_TO_GenericRobotOutputImage.Byte_[29]:= Motoman32_Typed_Data.IG30;
			FUN_GTAC_MOTOMAN32_TO_GenericRobotOutputImage.Byte_[30]:= Motoman32_Typed_Data.IG31;
			FUN_GTAC_MOTOMAN32_TO_GenericRobotOutputImage.Byte_[31]:= Motoman32_Typed_Data.IG32;
			FUN_GTAC_MOTOMAN32_TO_GenericRobotOutputImage.Byte_[32]:= Motoman32_Typed_Data.IG33;

END_FUNCTION

// ---- POUs/FBs/FB_GTAC_ProcessInterlock_20210526.TcPOU
(*
------------------------------------------------------------------------------------------
REVISION NOTES:
	Version 20210503
		- intial concept, j.underhill
	Version 20210526
		- added changed QA Reset to have Complete and Restart functionality
		- added Time Capture for Bypass activation
------------------------------------------------------------------------------------------
*)


FUNCTION_BLOCK FB_GTAC_ProcessInterlock_20210526
VAR_INPUT
	QA_Restart: BOOL;			(*FB Input to Force Restart of Interlocked Process*)
	QA_Complete: BOOL;			(*FB Input to Force Complete of Interlocked Process*)
	QA_Bypass: BOOL;			(*FB Input to Bypass Process Interlock by Quality*)

	Machine_Time: TimeStruct;	(*FB Input to Capture Time of Bypass*)

	Process_Started: BOOL;		(*FB Input to Capture Conditions to Start the Interlocked Process*)
	Offline_Process: BOOL;		(*FB Input to Capture Offline Process has Occured between Process Start and Complete*)
	Process_Completed: BOOL;	(*FB Input to Capture Conditions to Finish the Interlocked Process*)

END_VAR

VAR
	Bypass_TRIG: R_TRIG;		(*One Shot for Capture of Bypass Time*)
END_VAR

VAR PERSISTENT
	InProcess: BOOL;			(*Bit to Capture In Process*)
	OfflineProcess: BOOL;		(*Bit to Capture Offline Process*)
	PrevProcess: BOOL;			(*Bit for Previous Process Interlock*)
	NextProcess: BOOL;			(*Bit for Next Process Interlock*)
	Bypass_Time: TimeStruct;	(*FB Output to Indicate Time that Bypass was applied*)
END_VAR


VAR_OUTPUT
	Allow_PrevProcess: BOOL;	(*FB Output to Interlock with Prev Process to Continue*)
	Allow_NextProcess: BOOL;	(*FB Output to Interlock with Next Process to Continue*)

END_VAR

(*Capture In Process - Active From Process Started UNTIL Process Completed*)
	IF Process_Started OR QA_Restart
		THEN InProcess:= TRUE;
	ELSIF Process_Completed OR QA_Bypass
		THEN InProcess:= FALSE;
	END_IF;

(*Capture Offline Process - Active From Offline Process UNTIL Process Completed*)
	IF (InProcess AND Offline_Process) OR QA_Restart
		THEN OfflineProcess:= TRUE;
	ELSIF Process_Completed AND NOT Offline_Process
		THEN OfflineProcess:= FALSE;
	END_IF;

(*Allow Previous Process - Active From Process Completed UNTIL Process Started*)
	IF Process_Completed OR QA_Complete
		THEN PrevProcess:= TRUE;
	ELSIF InProcess OR OfflineProcess
		THEN PrevProcess:= FALSE;
	END_IF;
	Allow_PrevProcess:= PrevProcess OR QA_Bypass;

(*Allow Next Process - Active From Offline Process UNTIL Process Completed*)
	IF OfflineProcess
		THEN NextProcess:= TRUE;
	ELSIF (Process_Completed OR QA_Restart)
		THEN NextProcess:= FALSE;
	END_IF;
	Allow_NextProcess:= NextProcess OR QA_Bypass;


(*Capture Bypass Time*)
	Bypass_TRIG.CLK:= QA_Bypass;
	Bypass_TRIG();
	IF Bypass_TRIG.Q
		THEN Bypass_Time:= Machine_Time;
	END_IF;

END_FUNCTION_BLOCK

// ---- POUs/FBs/FB_GTAC_Reamer_20180405.TcPOU
(*FB for use with Mig Robot Tip Reamers

	Original Author(s): Brent Lekx-Toniolo of Sodecia GTAC.; 
------------------------------------------------------------------------------------------
REVISION NOTES:
	Version 20160210
		- intial concept, b.lekx-toniolo
	Version 20160831
		- added inputs and outputs for reaming, jvd
		-developed code to ream, jvd
	Version 20170327
		- added selection for Binzel/Fronius selection., j.vandongen
	Version 20170525
		- Cycle Correction for the Fronius., A. Lopez
	Version 20170531
		- Cycle Complete Correction for the Fronius. It sees the Cylinder Sensor too Quick. Added a Delay for the Cycle Completion., A. Lopez
	Version 20180405
		- changed N20 to N30 to follow new standards.
------------------------------------------------------------------------------------------
*)



FUNCTION_BLOCK FB_GTAC_Reamer_20180405

VAR_INPUT
	Enable_FB: BOOL;
	Enable_Motion: BOOL;

	Fronius_Ream: BOOL;
	Binzel_Ream: BOOL;

	WireCutter_REQ: BOOL;
	Injector_REQ: BOOL;
	Lift_REQ: BOOL;
	Clamp_REQ: BOOL;

	Ream_REQ: BOOL;
	Ream_Time: TIME;

END_VAR

VAR
(*Hardware Related Data Types*)
			(*Develop "Beckhoff Nodes"*)
			N01 AT %I*: udt_EP1008_002_v2;
			N30 AT %Q*: udt_EP2028_002_v2;
			N30_STAT AT %I*: udt_EP2028_002_STAT;

(* Nodes States*)
	DiscreteNode_OK: BOOL;
(* Cabel Break States*)
	ECatSlave_Cable_Breaks: UDINT;

	Ream_Step: UINT;
	LifterDown: BOOL;
	Clamp_Delay: TON;
	Ream_Delay: TON;
	Injector_Delay: TON;
	WireCutter_Delay: TON;
	LifterUp_Delay: TON;
	Reaming_Complete_Delay: TON;

END_VAR

VAR_OUTPUT

		FB_OK: BOOL;
		Discrete_Image: udt_Reamerxx_Image_20180405;

		LifterUp_ACK: BOOL;
		Clamp_ACK: BOOL;
		Injector_ACK: BOOL;
		WireCutter_ACK: BOOL;
		Reaming_Complete: BOOL;
END_VAR

	(*Set FB_OK to True*)
	FB_OK:= TRUE;

(*$$$$$$$$$$$$$$$$$$$$$$$$$$$$$$$$$$$$$$$$$$$$$$$$Gather Status Of Hardware $$$$$$$$$$$$$$$$$$$$$$$$$$$$$$$$$$$$$$$$$$$$$$$$$$$$*)
	(*Discrete I/O Nodes*)

	IF N01.InfoData.State=8 AND N30_STAT.InfoData.State=8
		THEN
			DiscreteNode_OK:=TRUE;
	ELSE
			DiscreteNode_OK:=FALSE;

	END_IF;

	(*Cable Break Detection*)
	ECatSlave_Cable_Breaks:= FUN_GTAC_EcatSlaveConnState
							(N01.InfoData.State,
							N30_STAT.InfoData.State,
							0,0,0,0,0,0,0,0,0,0,0,0,0,0,0,0,0,0,0,0,0,0,0,0,0,0,0,0); (*Function Returns Flags to warn of possible cable break*)



(*$$$$$$$$$$$$$$$$$$$$$$$$$$$$$$$$$$$$$$$$$$$$$$ Transfer Standard Outputs $$$$$$$$$$$$$$$$$$$$$$$$$$$$$$$$$$$$$$$$$$$*)
	(*Transfer I/O Images for Display On UI (User Interface)*)
	Discrete_Image.N01:=N01;
	Discrete_Image.N30:=N30;
	Discrete_Image.N30_STAT:=N30_STAT;

	Discrete_Image.ECatSlave_Cable_Breaks:= ECatSlave_Cable_Breaks;


(*????????????????????????????????????????????????? Develop Reaming Sequence Interlocks ???????????????????????????????????????????????????????????????*)

	IF Fronius_Ream (*Fronius Ream Selected*)
		THEN
			IF Reaming_Complete_Delay.Q
				THEN
					Reaming_Complete:= TRUE;
			ELSIF NOT Ream_Req
				THEN
					Reaming_Complete:=FALSE;
			END_IF;

			(*Fronius Cycle Complete Delay Timer*)
			Reaming_Complete_Delay(
					IN:= Ream_Req AND Ream_Delay.Q AND N01.I.0,
					PT:= T#1s,
					Q=> ,
					ET=> );

			(*Reaming Delay Timer*)
			Ream_Delay(
					IN:= Ream_Req,
					PT:= Ream_Time,
					Q=> ,
					ET=> );

			(*Reaming Output*)
			N30.Q.0:= Ream_Req AND NOT Ream_Delay.Q;


	ELSIF Binzel_Ream (*Binzel Ream Selected*)
		THEN
			(*Reaming Step 1 - Clamp*)
			Ream_Step.0 := Enable_Motion AND Ream_REQ AND NOT Reaming_Complete;

			(*Reaming Step 2 - Lifter*)
			Ream_Step.1 := Enable_Motion AND Ream_REQ AND NOT Reaming_Complete AND Clamp_Delay.Q;

			(*Ream_Step 3 - Lifter Down*)
			Ream_Step.2 := Enable_Motion AND Ream_REQ AND NOT Reaming_Complete AND Ream_Delay.Q;

			(*Ream_Step 4 - Clamp Release *)
			Ream_Step.3 := Enable_Motion AND Ream_REQ AND Reaming_Complete;

			(*Clamp Delay Timer*)
			Clamp_Delay(
					IN:= Ream_Step.0 OR Clamp_REQ,
					PT:= T#1s,
					Q=> ,
					ET=> );

			(*Reaming Delay Timer*)
			Ream_Delay(
					IN:= Ream_Step.1,
					PT:= Ream_Time,
					Q=> ,
					ET=> );

			(*Injector Delay Timer*)
			Injector_Delay(
					IN:= Injector_REQ,
					PT:= T#0.5s,
					Q=> ,
					ET=> );

			(*Cut Delay*)
			WireCutter_Delay(
					IN:= WireCutter_REQ,
					PT:= T#1s,
					Q=> ,
					ET=> );

			(*Lifter Up Delay*)
			LifterUp_Delay(
					IN:= NOT LifterDown,
					PT:= T#1s,
					Q=> ,
					ET=> );

			(*Lifter Down*)
			LifterDown:=N01.I.0;

			(*Lifter Up Ack*)
			 LifterUp_ACK:= LifterUp_Delay.Q;

			(*Clamp Ack*)
			Clamp_ACK := (Ream_REQ OR Clamp_REQ) AND Clamp_Delay.Q;

			(*Ream Complete ACK*)
			IF Ream_REQ AND NOT LifterUp_ACK AND Ream_Step.2
				THEN
				Reaming_Complete := TRUE;
			END_IF;

			IF Reaming_Complete AND NOT Ream_REQ
				THEN
				Reaming_Complete := FALSE;
			END_IF;

			(*Injector ACK*)
			Injector_ACK:= Injector_REQ AND Injector_Delay.Q;

			(*Wire Cutter ACK*)
			WireCutter_ACK:= WireCutter_REQ AND WireCutter_Delay.Q;

			(*Wire Cutter*)
			N30.Q.0 := WireCutter_REQ AND NOT WireCutter_Delay.Q;

			(*Injector*)
			N30.Q.1:= Injector_REQ AND NOT Injector_Delay.Q;

			(*Lift*)
			N30.Q.2:=Lift_REQ OR (Ream_Step.1AND NOT Ream_Step.2 AND NOT Ream_Step.3);

			(*Clamp*)
			N30.Q.3:= Clamp_REQ OR ((Ream_Step.0 OR Ream_Step.1 OR Ream_Step.2) AND NOT Ream_Step.3);
	END_IF;




(*end*)

END_FUNCTION_BLOCK

// ---- POUs/FBs/FB_Model_Status.TcPOU
(*FB for ???:
	Original Author(s): ??? 
	August 2010; version 3.0*)

FUNCTION_BLOCK FB_Model_Status

	VAR_INPUT
		Enable_FB: BOOL;
		Enable_LookFor_Hole: BOOL;
		Found_Metal_Sensor: BOOL;
		Found_Hole_Sensor: BOOL;
		Retracted_Sensor: BOOL;
		Advance_Solenoid: BOOL;
		Retract_Solenoid: BOOL;
		Metal_Delay: TIME;
		Hole_Delay: TIME;
		Ret_Delay: TIME;
		Fault_Delay: TIME;
	END_VAR

	VAR
		At_Metal: BOOL;
		At_Hole: BOOL;
		At_Retracted: BOOL;
		Metal_Delay_TMR: TON;
		Hole_Delay_TMR: TON;
		Ret_Delay_TMR: TON;
		Sensor_FLT_TMR: TON;
		Advancing_FLT_TMR: TON;
		Retracting_FLT_TMR: TON;
	END_VAR

	VAR_OUTPUT
		FB_OK: BOOL;
		In_Metal_Position: BOOL;
		In_Hole_Position: BOOL;
		In_Retracted_Position: BOOL;
		Faulted: BOOL;
		Sensor_Fault: BOOL;
		Advancing_Fault: BOOL;
		Retracting_Fault: BOOL;
	END_VAR

	(*Set FB_OK to True*)
	FB_OK:= TRUE;
(*$$$$$$$$$$$$$$$$$$$$$$$$$$$$$$$$$$ Internal Code $$$$$$$$$$$$$$$$$$$$$$$$$$$$$$$$$$$$$$$$$$$$$$$*)
	(*Develop Metal Position*)
	At_Metal:=Found_Metal_Sensor AND NOT Retracted_Sensor;
	(*Develop Hole Position*)
	At_Hole:=Found_Hole_Sensor AND NOT Retracted_Sensor;

	(*Develop Retracted Position*)
	At_Retracted:=Retracted_Sensor AND NOT Found_Metal_Sensor AND NOT Found_Hole_Sensor;

	(*Delay Metal  Position Output*)
	Metal_Delay_TMR.PT:=Metal_Delay;
	Metal_Delay_TMR.IN:=At_Metal;
	Metal_Delay_TMR();
	In_Metal_Position:=Metal_Delay_TMR.Q;

	(*Delay Hole  Position Output*)
	Hole_Delay_TMR.PT:=Hole_Delay;
	Hole_Delay_TMR.IN:=At_Hole;
	Hole_Delay_TMR();
	In_Hole_Position:=Hole_Delay_TMR.Q;

	(*Delay Retracted Position Output*)
	Ret_Delay_TMR.PT:=Ret_Delay;
	Ret_Delay_TMR.IN:=At_Retracted;
	Ret_Delay_TMR();
	In_Retracted_Position:=Ret_Delay_TMR.Q;

(*$$$$$$$$$$$$$$$$$$$$$$$$$$$$$$$$$$$$$$$$ Fault Code $$$$$$$$$$$$$$$$$$$$$$$$$$$$$$$$$$$$$$$$$$$$$$$$*)
	(*Sensor Fault*)
	Sensor_FLT_TMR.PT:=Fault_Delay;
	Sensor_FLT_TMR.IN:=(NOT At_Metal AND NOT At_Hole AND NOT At_Retracted) OR (At_Metal AND At_Retracted) OR (At_Hole AND At_Retracted) OR (At_Metal AND At_Hole);
	Sensor_FLT_TMR();
	Sensor_Fault:=Sensor_FLT_TMR.Q;

	(*Advancing Fault*)
	Advancing_FLT_TMR.PT:=Fault_Delay;
	Advancing_FLT_TMR.IN:=Advance_Solenoid AND (NOT At_Metal OR NOT At_Hole) AND NOT Sensor_Fault;
	Advancing_FLT_TMR();
	Advancing_Fault:=Advancing_FLT_TMR.Q;

	(*Retracting Fault*)
	Retracting_FLT_TMR.PT:=Fault_Delay;
	Retracting_FLT_TMR.IN:=Retract_Solenoid AND NOT At_Retracted AND NOT Sensor_Fault;
	Retracting_FLT_TMR();
	Retracting_Fault:=Retracting_FLT_TMR.Q;

	(*Develop Fault Output*)
	Faulted:= Sensor_Fault OR Advancing_Fault OR Retracting_Fault;

END_FUNCTION_BLOCK

// ---- POUs/FBs/FB_UDP_PortCreate20140120.TcPOU
FUNCTION_BLOCK FB_UDP_PortCreate20140120
VAR_INPUT

	LocalNetID:						STRING(19);
	Local_IP_Address:				STRING(15);
	UDP_Port_Number:				UINT;
	ConnectUdp:						BOOL;
	CloseUdp:						BOOL;

END_VAR
VAR_OUTPUT

	UdpSocketHandle:				T_HSocket;									(*Open Udp Socket Connection Information*)
	Port_Closed:						BOOL;										(*Socket Close has been executed*)
	UdpReceiveLength:				UDINT;
	UdpReceived:					STRING;

END_VAR
VAR
(*Required Udp variables*)
	SocketUdpCreate:					FB_SocketUdpCreate;							(*Opens the Udp Socket in the Local Controller*)
	SocketClose:						FB_SocketClose;								(*Closes the Udp Socket*)
	SocketUdpReceiveFrom:			FB_SocketUdpReceiveFrom;					(*Gathers Received Data from all devices*)

	pDest:							POINTER TO STRING;

END_VAR

VAR CONSTANT



END_VAR

pDest := ADR(UdpReceived);										(*Point to address of variable to store reply data*)






(*---------------------------------------------------------FB Instances------------------------------------------------------*)


(*UDP Socket creation for Config Data*)
SocketUdpCreate(
	sSrvNetId:= LocalNetID,
	sLocalHost:=Local_IP_Address,
	nLocalPort:= UDP_Port_Number,
	bExecute:= ConnectUdp,
	tTimeout:= T#50s,
	bBusy=> ,
	bError=> ,
	nErrId=> ,
	hSocket=> UdpSocketHandle);


(*UDP Socket Close*)
SocketClose(
	sSrvNetId:= LocalNetID,
	hSocket:= UdpSocketHandle,
	bExecute:= CloseUdp,
	tTimeout:= T#5s,
	bBusy=> ,
	bError=> ,
	nErrId=> );

IF CloseUdp
	THEN
		Port_Closed:=TRUE;
ELSE
		Port_Closed:= FALSE;
END_IF;

(*UDP Receive Function Block*)
SocketUdpReceiveFrom(
	sSrvNetId:= LocalNetID,
	hSocket:= UdpSocketHandle,
	cbLen:= 80,
	pDest:= pDest,
	bExecute:= Pulse_500ms,
	tTimeout:= T#30s,
	bBusy=> ,
	bError=> ,
	nErrId=> ,
	sRemoteHost=> ,
	nRemotePort=> ,
	nRecBytes=> UdpReceiveLength);

END_FUNCTION_BLOCK

// ---- POUs/FUNs/FUN_GTAC_DINTtoINT.TcPOU
(*Copies and truncates a DINT (input to the FUN) at bit level, into individual bits of the INT Return, based upon a byte shift index intput
Valid Byte Shift Input values is 0-3

	author: Brent Lekx-Toniolo OF Sodecia GTAC
	date: Sept 2015
	version 1.0
		- initial concept
	Last Edit: 29-Sept-2015, BLT
*)

FUNCTION FUN_GTAC_DINTtoINT : INT
VAR_INPUT
	Dint0: DINT;
	Byte_Shift_Index: UINT;
END_VAR
VAR
END_VAR

(*Copy Bytes from DINT to INT return, based upon Byte Shift Index*)

IF Byte_Shift_Index=0
	THEN
	(*Byte Shift Index of 0, staright copy first two bytes of Dint to Return*)
	FUN_GTAC_DINTtoINT.0:= Dint0.0;
	FUN_GTAC_DINTtoINT.1:= Dint0.1;
	FUN_GTAC_DINTtoINT.2:= Dint0.2;
	FUN_GTAC_DINTtoINT.3:= Dint0.3;
	FUN_GTAC_DINTtoINT.4:= Dint0.4;
	FUN_GTAC_DINTtoINT.5:= Dint0.5;
	FUN_GTAC_DINTtoINT.6:= Dint0.6;
	FUN_GTAC_DINTtoINT.7:= Dint0.7;

	FUN_GTAC_DINTtoINT.8:= Dint0.8;
	FUN_GTAC_DINTtoINT.9:= Dint0.9;
	FUN_GTAC_DINTtoINT.10:= Dint0.10;
	FUN_GTAC_DINTtoINT.11:= Dint0.11;
	FUN_GTAC_DINTtoINT.12:= Dint0.12;
	FUN_GTAC_DINTtoINT.13:= Dint0.13;
	FUN_GTAC_DINTtoINT.14:= Dint0.14;
	FUN_GTAC_DINTtoINT.15:= Dint0.15;

ELSIF Byte_Shift_Index=1
	THEN
	(*Byte Shift Index of 1, copy from Dint byte1 to Return*)
	FUN_GTAC_DINTtoINT.0:= Dint0.8;
	FUN_GTAC_DINTtoINT.1:= Dint0.9;
	FUN_GTAC_DINTtoINT.2:= Dint0.10;
	FUN_GTAC_DINTtoINT.3:= Dint0.11;
	FUN_GTAC_DINTtoINT.4:= Dint0.12;
	FUN_GTAC_DINTtoINT.5:= Dint0.13;
	FUN_GTAC_DINTtoINT.6:= Dint0.14;
	FUN_GTAC_DINTtoINT.7:= Dint0.15;

	FUN_GTAC_DINTtoINT.8:= Dint0.16;
	FUN_GTAC_DINTtoINT.9:= Dint0.17;
	FUN_GTAC_DINTtoINT.10:= Dint0.18;
	FUN_GTAC_DINTtoINT.11:= Dint0.19;
	FUN_GTAC_DINTtoINT.12:= Dint0.20;
	FUN_GTAC_DINTtoINT.13:= Dint0.21;
	FUN_GTAC_DINTtoINT.14:= Dint0.22;
	FUN_GTAC_DINTtoINT.15:= Dint0.23;

ELSIF Byte_Shift_Index=2
	THEN
	(*Byte Shift Index of 2, copy from Dint byte2 to Return*)
	FUN_GTAC_DINTtoINT.0:= Dint0.16;
	FUN_GTAC_DINTtoINT.1:= Dint0.17;
	FUN_GTAC_DINTtoINT.2:= Dint0.18;
	FUN_GTAC_DINTtoINT.3:= Dint0.19;
	FUN_GTAC_DINTtoINT.4:= Dint0.20;
	FUN_GTAC_DINTtoINT.5:= Dint0.21;
	FUN_GTAC_DINTtoINT.6:= Dint0.22;
	FUN_GTAC_DINTtoINT.7:= Dint0.23;

	FUN_GTAC_DINTtoINT.8:= Dint0.24;
	FUN_GTAC_DINTtoINT.9:= Dint0.25;
	FUN_GTAC_DINTtoINT.10:= Dint0.26;
	FUN_GTAC_DINTtoINT.11:= Dint0.27;
	FUN_GTAC_DINTtoINT.12:= Dint0.28;
	FUN_GTAC_DINTtoINT.13:= Dint0.29;
	FUN_GTAC_DINTtoINT.14:= Dint0.30;
	FUN_GTAC_DINTtoINT.15:= Dint0.31;

ELSIF Byte_Shift_Index=3
	THEN
	(*Byte Shift Index of 3, copy from Dint byte3 to Return and blank unused byte in return*)
	FUN_GTAC_DINTtoINT.0:= Dint0.24;
	FUN_GTAC_DINTtoINT.1:= Dint0.25;
	FUN_GTAC_DINTtoINT.2:= Dint0.26;
	FUN_GTAC_DINTtoINT.3:= Dint0.27;
	FUN_GTAC_DINTtoINT.4:= Dint0.28;
	FUN_GTAC_DINTtoINT.5:= Dint0.29;
	FUN_GTAC_DINTtoINT.6:= Dint0.30;
	FUN_GTAC_DINTtoINT.7:= Dint0.31;

	FUN_GTAC_DINTtoINT.8:= FALSE;
	FUN_GTAC_DINTtoINT.9:= FALSE;
	FUN_GTAC_DINTtoINT.10:= FALSE;
	FUN_GTAC_DINTtoINT.11:= FALSE;
	FUN_GTAC_DINTtoINT.12:= FALSE;
	FUN_GTAC_DINTtoINT.13:= FALSE;
	FUN_GTAC_DINTtoINT.14:= FALSE;
	FUN_GTAC_DINTtoINT.15:= FALSE;

ELSE
	(*default case, blank return*)
	FUN_GTAC_DINTtoINT.0:= FALSE;
	FUN_GTAC_DINTtoINT.1:= FALSE;
	FUN_GTAC_DINTtoINT.2:= FALSE;
	FUN_GTAC_DINTtoINT.3:= FALSE;
	FUN_GTAC_DINTtoINT.4:= FALSE;
	FUN_GTAC_DINTtoINT.5:= FALSE;
	FUN_GTAC_DINTtoINT.6:= FALSE;
	FUN_GTAC_DINTtoINT.7:= FALSE;

	FUN_GTAC_DINTtoINT.8:= FALSE;
	FUN_GTAC_DINTtoINT.9:= FALSE;
	FUN_GTAC_DINTtoINT.10:= FALSE;
	FUN_GTAC_DINTtoINT.11:= FALSE;
	FUN_GTAC_DINTtoINT.12:= FALSE;
	FUN_GTAC_DINTtoINT.13:= FALSE;
	FUN_GTAC_DINTtoINT.14:= FALSE;
	FUN_GTAC_DINTtoINT.15:= FALSE;

END_IF;

END_FUNCTION

// ---- POUs/FUNs/FUN_GTAC_FindStringInArray.TcPOU
(*Function to return a portion of source string (from a provided string) based on return length specified (starting at element 0 of source)
	author: Brent Lekx-Toniolo OF Sodecia GTAC
	date: May 2016
	version 1.0
		- initial concept
	Last Edit: 11-May-2016, 
		- create FUN, blt

*)


FUNCTION FUN_GTAC_FindStringInArray : UINT
VAR_INPUT
	Search_String: STRING[5];											(*String to Search for*)
	ptrArray_To_Search: POINTER TO ARRAY[0..100] OF STRING [5];		(*Pointer to Array to Search through*)
END_VAR

VAR
	Search_Index: UINT;
END_VAR

(*-------------------------------------- Search through Array Passed for String -----------------------------------*)

	FOR Search_Index:= 0 TO 99 DO
		IF (ptrArray_To_Search^[Search_Index]= Search_String)		(*Dereference (^) pointer in order to access the data in the object referenced by pointer, then compare to the string being requested*)
			THEN
			FUN_GTAC_FindStringInArray:= Search_Index;			(*Capture Array Location*)
		END_IF;

	END_FOR;

END_FUNCTION

// ---- POUs/FUNs/FUN_GTAC_GetNodeFromName.TcPOU
FUNCTION FUN_GTAC_GetNodeFromName : String
VAR_INPUT
	InputString:STRING;
	
END_VAR
VAR
	SpaceLoc :INT;
	PeriodLoc:INT;
END_VAR


(*Find the '.' location in the input string *)
PeriodLoc := find(InputString,'.');
SpaceLoc := find(InputString,' ');

(*Using the above location, cut the name out of the input string, and return that as our string*)
IF (SpaceLoc - PeriodLoc) = 5 THEN
	FUN_GTAC_GetNodeFromName:= mid(InputString,4,PeriodLoc+1);
ELSE
	FUN_GTAC_GetNodeFromName:= mid(InputString,3,PeriodLoc+1);
END_IF

END_FUNCTION

// ---- POUs/FUNs/FUN_GTAC_OTSTRUCTtoTOD.TcPOU
(*Take Individual time elements of a OTSTRUCT and create a TOD type return
	author: Brent Lekx-Toniolo Of Sodecia GTAC
	date: May 2016
	version 1.0
		- initial concept


	Last Edit: 27-May-2016, blt
*)

FUNCTION FUN_GTAC_OTSTRUCTtoTOD : TOD
VAR_INPUT
	OTSTRUCT: OTSTRUCT;

END_VAR
VAR
	Hours_as_MS: UDINT;
	Minutes_as_MS: UDINT;
	Seconds_as_MS: UDINT;
	Milliseconds_as_MS: UDINT;
END_VAR

(*Calculate Millsecond Value of each OTSTRUCT Element*)

	Hours_as_MS:= OTSTRUCT.wHour * 360000;
	Minutes_as_MS:= OTSTRUCT.wMinute * 60000;
	Seconds_as_MS:= OTSTRUCT.wSecond * 1000;
	Milliseconds_as_MS:= OTSTRUCT.wMilliseconds;

(*Return Total Value in Milliseconds, this is TOD*)

FUN_GTAC_OTSTRUCTtoTOD:= UDINT_TO_TOD(Hours_As_MS + Minutes_As_MS + Seconds_As_MS + Milliseconds_As_MS);

END_FUNCTION

// ---- POUs/FUNs/FUN_GTAC_OTSTRUCTWrapper.TcPOU
(*Copy Individual data elements into an OTSTRUCT TYPE
	author: Brent Lekx-Toniolo Of Sodecia GTAC
	date: May 2016
	version 1.0
		- initial concept


	Last Edit: 19-May-2016, blt
*)



FUNCTION FUN_GTAC_OTSTRUCTWrapper : OTSTRUCT
VAR_INPUT
	(*NOTE: WEEK, DAY and MILLISEC not used in this wrapper*)
	(*
	Week: WORD;
	Day: WORD;
	*)
	Hour: WORD;
	Minute: WORD;
	Second: WORD;
			(*
	Milliseconds: WORD;
	*)

END_VAR

VAR
END_VAR

(*Retrieve Data, Load to Return Type*)

	FUN_GTAC_OTSTRUCTWrapper.wWeek:= 0;
	FUN_GTAC_OTSTRUCTWrapper.wDay:= 0;
	FUN_GTAC_OTSTRUCTWrapper.wHour:= Hour;
	FUN_GTAC_OTSTRUCTWrapper.wMinute:= Minute;
	FUN_GTAC_OTSTRUCTWrapper.wSecond:= Second;
	FUN_GTAC_OTSTRUCTWrapper.wMilliseconds:= 0;

END_FUNCTION

// ---- POUs/FUNs/FUN_RailMove_To_ICxx.TcPOU
FUNCTION FUN_RailMove_To_ICxx : REAL
FUNCTION FUN_Railmove_To_ICxx : REAL;
VAR_INPUT
    InValue   : INT;   // Based on Sim  Robot Axis value (-15700 … +200) 
    P_Min    : REAL;   // Page min (e.g. 550)
    P_Max    : REAL;   // Page max (e.g. 750)
	R_Min     : REAL;  //  axis min of the robot on each line overview
    R_MAX     : REAL;  //  axis max of the robot on each line overview
END_VAR
 
VAR
    ScaleFactor : REAL;
END_VAR



ScaleFactor := (P_Max - P_Min) / (R_Max - R_Min);
FUN_Railmove_To_ICxx := (InValue - R_Min) * ScaleFactor + P_Min;

END_FUNCTION
